(*
SPDX-FileCopyrightText: © 2026 Oleksandr Tiutyk <trofimich@gmail.com>
SPDX-License-Identifier: MIT
License: https://opensource.org/license/mit
*)

INTERFACE IEventDispatcher EXTENDS IBubbleEventDispatcher, IBroadcastEventDispatcher

END_INTERFACE

(* stored: Version 1.1.0.1
   Itf IEventDispatcher: Id {8298e301-c120-44f5-89f7-9228bd80d23e} *)
